(*			
	EVERDE sp. z o.o.
	Rafał Osajda		08.08.2025		TC 4024.66
	Interfejs do wyciągania z SPM przez HMI danych do wyświetlania - dla ramki głównej tryp pracy konserwacja
*)
INTERFACE ITF_SPM_HMI_00_02_Lacznik EXTENDS  B_Baza.ITF_ZrodloIdentyfikacji

END_INTERFACE

(* stored: Version 1.1.0.1
   Itf ITF_SPM_HMI_00_02_Lacznik: Id {20ffc7a6-37bd-0c7f-1b58-7ddf3bf9f8a7} *)
